FUNCTION_BLOCK WP_Sensor (* Composite Function Block Type *)
  (* Standard: 61499-2 *)
  (* Version 0.0, 2/7/2012, XPMUser, nxtControl GmbH, template *)
  PACKAGE Main;
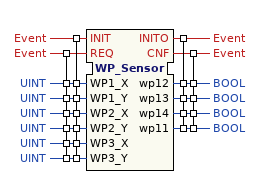
  EVENT_INPUT
    INIT WITH WP1_X, WP1_Y, WP2_X, WP2_Y, WP3_Y, WP3_X; (* Initialization Request *)
    REQ WITH WP1_Y, WP1_X, WP2_X, WP2_Y, WP3_X, WP3_Y; (* Normal Execution Request *)
  END_EVENT
  EVENT_OUTPUT
    INITO WITH wp12, wp14, wp11, wp13; (* Initialization Confirm *)
    CNF WITH wp12, wp13, wp14, wp11; (* Execution Confirmation *)
  END_EVENT
  VAR_INPUT
    WP1_X : UINT;
    WP1_Y : UINT;
    WP2_X : UINT;
    WP2_Y : UINT;
    WP3_X : UINT;
    WP3_Y : UINT;
  END_VAR
  VAR_OUTPUT
    wp12 : BOOL;
    wp13 : BOOL;
    wp14 : BOOL;
    wp11 : BOOL;
  END_VAR
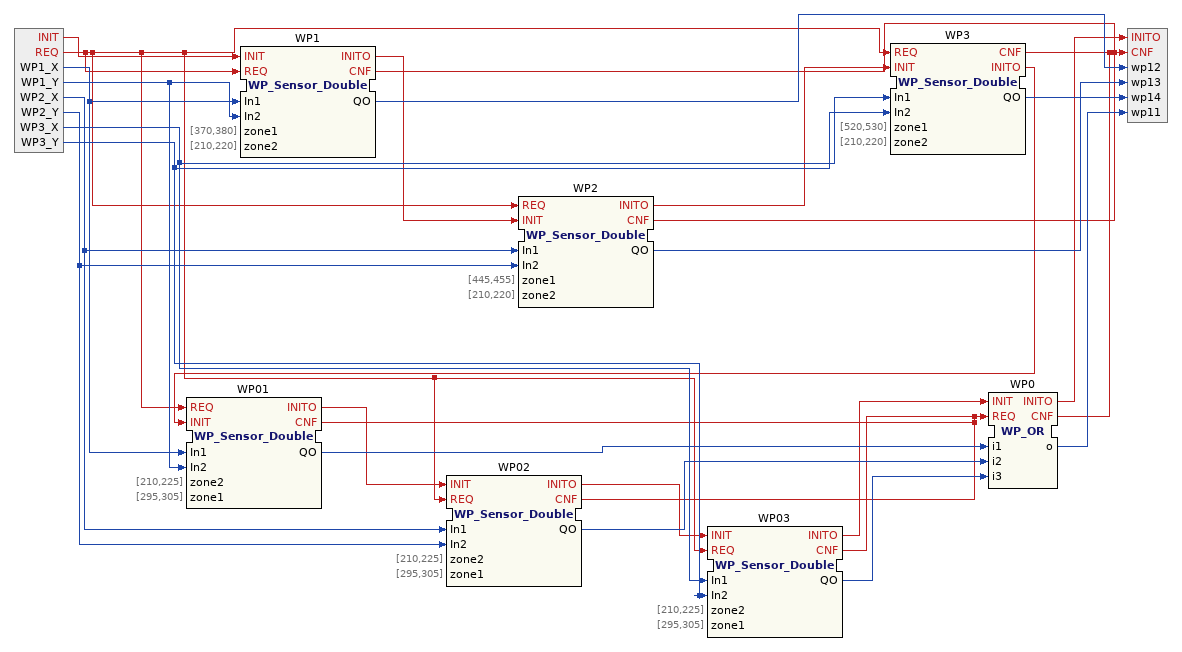
  FBS
    WP1 : WP_Sensor_Double(zone1 := [370,380], zone2 := [210,220]);
    WP2 : WP_Sensor_Double(zone1 := [445,455], zone2 := [210,220]);
    WP3 : WP_Sensor_Double(zone1 := [520,530], zone2 := [210,220]);
    WP01 : WP_Sensor_Double(zone2 := [210,225], zone1 := [295,305]);
    WP02 : WP_Sensor_Double(zone2 := [210,225], zone1 := [295,305]);
    WP03 : WP_Sensor_Double(zone2 := [210,225], zone1 := [295,305]);
    WP0 : WP_OR;
  END_FBS
  EVENT_CONNECTIONS
    INIT TO WP1.INIT;
    REQ TO WP1.REQ;
    REQ TO WP2.REQ;
    REQ TO WP3.REQ;
    WP1.INITO TO WP2.INIT;
    WP2.INITO TO WP3.INIT;
    WP1.CNF TO CNF;
    WP2.CNF TO CNF;
    WP3.CNF TO CNF;
    REQ TO WP01.REQ;
    WP01.INITO TO WP02.INIT;
    WP02.INITO TO WP03.INIT;
    REQ TO WP02.REQ;
    REQ TO WP03.REQ;
    WP03.INITO TO WP0.INIT;
    WP03.CNF TO WP0.REQ;
    WP02.CNF TO WP0.REQ;
    WP01.CNF TO WP0.REQ;
    WP0.CNF TO CNF;
    WP0.INITO TO INITO;
    WP3.INITO TO WP01.INIT;
  END_CONNECTIONS
  DATA_CONNECTIONS
    WP1.QO TO wp12;
    WP2.QO TO wp13;
    WP3.QO TO wp14;
    WP1_X TO WP1.In1;
    WP1_Y TO WP1.In2;
    WP2_X TO WP2.In1;
    WP2_Y TO WP2.In2;
    WP3_X TO WP3.In1;
    WP3_Y TO WP3.In2;
    WP1_X TO WP01.In1;
    WP1_Y TO WP01.In2;
    WP2_X TO WP02.In1;
    WP2_Y TO WP02.In2;
    WP3_X TO WP03.In1;
    WP3_Y TO WP03.In2;
    WP03.QO TO WP0.i3;
    WP02.QO TO WP0.i2;
    WP01.QO TO WP0.i1;
    WP0.o TO wp11;
  END_CONNECTIONS
END_FUNCTION_BLOCK
